TYPE HMI_MAN_RbtFanucUnloading EXTENDS HMI_MAN_RbtFanuc:
STRUCT
	;//add custom bools on top of library block here
END_STRUCT
END_TYPE

(* stored: Version 1.1.0.1
   DUT HMI_MAN_RbtFanucUnloading: Id {71fa92c6-aa36-4e6b-ad75-b766a1a4998c} *)
